TYPE arr8Bit :
STRUCT
	data8Bit : ARRAY[0..7] OF BOOL;
END_STRUCT
END_TYPE

(* stored: Version 1.1.0.1, ProductVersion 3.1.4024.11
   DUT arr8Bit: Id {9af8f754-b85b-4ecc-9609-7b3988d475dc} *)
